// TIA Portal V16 export
// export: Created 2024-12-03T15:41:45.4146913Z, ExportSetting WithReadOnly, DisplayName Totally Integrated Automation Portal, DisplayVersion V16 Update 6, DisplayName TIA Portal Version Control Interface, DisplayVersion V16 Update 2, DisplayName TIA Portal Openness, DisplayVersion V16 Update 6, DisplayName TIA Portal Teamcenter Gateway, DisplayVersion V16, DisplayName SINAMICS Startdrive Advanced, DisplayVersion V16 Update 5, DisplayName SINAMICS Startdrive G130, G150, S120, S150, SINAMICS MV, S210, DisplayVersion V16 Update 5, DisplayName SINAMICS Startdrive G110M, G120, G120C, G120D, G120P, G115D, DisplayVersion V16 Update 5, DisplayName STEP 7 Professional, DisplayVersion V16 Update 6, DisplayName STEP 7 Safety, DisplayVersion V16, DisplayName WinCC Advanced / Unified PC, DisplayVersion V16 Update 6
TYPE "G115D_INPUT_UDT"
// stored: CreationDate 2022-02-10T10:30:20.6863124Z, InterfaceModifiedDate 2021-08-10T11:20:19.6458047Z, IsConsistent true, LibraryConformanceStatus The object is library-conformant., ModifiedDate 2021-08-10T11:20:19.6458047Z
   STRUCT
      status : Struct
         RunningAtSpeed : Bool;
         ControlRequest : Bool;
         MaxSpeedExceeded : Bool;
         TorQueOk : Bool;
         MotorHoldingBrakeOPen : Bool;
         TemperatureOk : Bool;
         MotorRotating : Bool;
         CurrentOk : Bool;
         readyForSwitchOn : Bool;
         Ready : Bool;
         OperationEnabled : Bool;
         FaultActive : Bool;
         CoastDownActive : Bool;
         QuickStopActive : Bool;
         InhibitedActive : Bool;
         AlarmActive : Bool;
      END_STRUCT;
      Speed : Word;
      Current : Word;
      Torque : Word;
      WarnCode : Word;
      FaultCode : Word;
      extension : "GXXX_EXTENSION_INPUT_UDT";
   END_STRUCT;
END_TYPE
